FUNCTION INTERNAL F_SbhRecomputeBufferSizeAfterLimit : HRESULT
VAR_IN_OUT
    stState     : ST_ParserInternalState;
END_VAR
VAR
    nBufferEnd  : UDINT;
END_VAR


stState.nBufferSize := stState.nBufferSize + stState.nBufferSizeAfterLimit;

nBufferEnd := stState.nTotalBytesRetired + stState.nBufferSize;

IF nBufferEnd > stState.nCurrentLimit THEN
    stState.nBufferSizeAfterLimit := nBufferEnd - stState.nCurrentLimit;
    stState.nBufferSize := stState.nBufferSize - stState.nBufferSizeAfterLimit;
ELSE
    stState.nBufferSizeAfterLimit := 0;
END_IF

END_FUNCTION

(* stored: Version 1.1.0.1
   POU F_SbhRecomputeBufferSizeAfterLimit: Id {15ebdb48-aded-44d6-a039-ca8ad43032c4}, SpecialFunc None *)
